FUNCTION_BLOCK FB_AlarmLogListener EXTENDS FB_FCSLBaseKeyValueLogListener

METHOD Initialize : BOOL
VAR
    ListenerFilter : FB_TcEventFilter;
    hr             : HRESULT;
END_VAR
Listener := THIS^;                                   //For callbacks on message received
ListenerFilter.Clear().EventClass.EqualTo(TC_EVENT_CLASSES.AlarmLog); //Filter events by tracing class
hr := Subscribe2(ListenerFilter);                    //Subscribe to retrieve defined events
IF ( SUCCEEDED(hr) ) THEN
    Initialize := TRUE;
END_IF
END_METHOD

END_FUNCTION_BLOCK

(* stored: Version 1.1.0.1
   POU FB_AlarmLogListener: Id {17741a68-c7bb-46f1-8c9b-fba3b3562d9d}, SpecialFunc None
   Method Initialize: Id {431a49c3-2e24-4c2c-b870-5e13e043c5c3} *)
